// TIA Portal project "Övning 5" (V16)

(* hardware
DEVICE "S7-1200 station_1"  S7-1200 Station
   slot 0: "Rack_0"  S7-1200 Rack  Rack  V1.0
   slot 1: "PLC_1"  CPU 1212C DC/DC/DC  6ES7 212-1AE40-0XB0  V4.2
   slot 2: "DI 16x24VDC_1"  6ES7 221-1BH32-0XB0  V2.0
   slot 3: "DQ 16x24VDC_1"  SM 1222 DQ16 x 24VDC  6ES7 222-1BH32-0XB0  V2.0
*)

// ===== PLC "PLC_1"  CPU 1212C DC/DC/DC =====

VAR_GLOBAL   // PLC tag table "Default tag table"
   "ÅTERSTÄLLNING" AT %I0.0 : Bool;
   "VRED_MANUEL" AT %I0.1 : Bool;
   "VRED_AUTO" AT %I0.2 : Bool;
   "K_START" AT %I0.3 : Bool;
   "K_STOPP" AT %I0.4 : Bool;
   "K_PUMP1_TILL" AT %I0.5 : Bool;
   "K_PUMP1_FRÅN" AT %I0.6 : Bool;
   "K_PUMP2_TILL" AT %I8.0 : Bool;
   "K_PUMP2_FRÅN" AT %I8.1 : Bool;
   "K_VENTIL_STÄNG" AT %I8.2 : Bool;
   "K_VENTIL_ÖPPNA" AT %I8.3 : Bool;
   "K_LAMPTEST" AT %I8.4 : Bool;
   "NIVÅ_L6" AT %I9.0 : Bool;
   "NIVÅ_L5" AT %I9.1 : Bool;
   "NIVÅ_L4" AT %I9.2 : Bool;
   "NIVÅ_L3" AT %I9.3 : Bool;
   "NIVÅ_L2" AT %I9.4 : Bool;
   "NIVÅ_L1" AT %I9.5 : Bool;
   "MOTORSKYDD_B1" AT %I9.6 : Bool;
   "MOTORSKYDD_F2" AT %I9.7 : Bool;
   "L_ALARM" AT %Q12.0 : Bool;
   "L_PUMP1_TILL" AT %Q12.1 : Bool;
   "L_PUMP1_FRÅN" AT %Q12.2 : Bool;
   "L_VENTIL_ÖPPEN" AT %Q12.3 : Bool;
   "L_VENTIL_STÄNGD" AT %Q12.4 : Bool;
   "L_PUMP2_TILL" AT %Q12.5 : Bool;
   "L_PUMP2_FRÅN" AT %Q12.6 : Bool;
   "L_NIVÅ_ALARM" AT %Q12.7 : Bool;
   "KONTAKTOR_H" AT %Q13.0 : Bool;
   "KONTAKTOR_D" AT %Q13.1 : Bool;
   "KONTAKTOR_Y" AT %Q13.2 : Bool;
   "KONTAKTOR_DIREKT" AT %Q13.3 : Bool;
   "KONTAKTOR_MAGNETVENTIL" AT %Q13.4 : Bool;
   "KONTAKTOR_IND.VENTIL" AT %Q13.5 : Bool;
   "KONTAKTOR_BLIXT" AT %Q13.6 : Bool;
   "M_AUTO" AT %M0.0 : Bool;
   "M_MANUELL" AT %M0.1 : Bool;
   "M_VENTIL_ÖPPNA/STÄNG_MANU" AT %M0.2 : Bool;
   "M_PUMP1_TILL_MANUELL" AT %M0.3 : Bool;
   "M_PUMP2_TILL_MANUELL" AT %M0.4 : Bool;
   "M_VENTIL_ÖPPNA/STÄNG_AUTO" AT %M0.5 : Bool;
   "M_PUMP1_TILL_AUTO" AT %M0.6 : Bool;
   "M_PUMP2_TILL_AUTO" AT %M0.7 : Bool;
   "M_VARRANAN" AT %M1.0 : Bool;
   "M_BLIXT_AUTO" AT %M1.1 : Bool;
   "M_LARM_NIVÅ_AUTO" AT %M1.2 : Bool;
   "System_Byte" AT %MB1 : Byte;
   "Clock_Byte" AT %MB500 : Byte;
   "Clock_10Hz" AT %M500.0 : Bool;
   "Clock_5Hz" AT %M500.1 : Bool;
   "Clock_2.5Hz" AT %M500.2 : Bool;
   "Clock_2Hz" AT %M500.3 : Bool;
   "Clock_1.25Hz" AT %M500.4 : Bool;
   "Clock_1Hz" AT %M500.5 : Bool;
   "Clock_0.625Hz" AT %M500.6 : Bool;
   "Clock_0.5Hz" AT %M500.7 : Bool;
   "M_LARM_BLINKIE" AT %M2.0 : Bool;
   "M_LAMPTEST" AT %M2.1 : Bool;
   "M_LAMPTEST_AUTO" AT %M2.2 : Bool;
END_VAR

// folder: System blocks/Program resources

DATA_BLOCK "TIMER Y/D"   // DB1
{ S7_Optimized_Access := 'TRUE' }
AUTHOR : Simatic
FAMILY : IEC
NAME : IEC_TMR
VERSION : 1.0
// stored: InstanceOfName IEC_TIMER
"IEC_TIMER"
BEGIN
END_DATA_BLOCK

DATA_BLOCK "BLIXT-TIMER"   // DB2
{ S7_Optimized_Access := 'TRUE' }
AUTHOR : Simatic
FAMILY : IEC
NAME : IEC_TMR
VERSION : 1.0
// stored: InstanceOfName IEC_TIMER
"IEC_TIMER"
BEGIN
END_DATA_BLOCK

DATA_BLOCK "LAMP_TEST_AUTO"   // DB3
{ S7_Optimized_Access := 'TRUE' }
AUTHOR : Simatic
FAMILY : IEC
NAME : IEC_TMR
VERSION : 1.0
// stored: InstanceOfName IEC_TIMER
"IEC_TIMER"
BEGIN
END_DATA_BLOCK

// folder: (top level)

FUNCTION "Mongo" : Void   // FC1, LAD
{ S7_Optimized_Access := 'TRUE' }
VERSION : 0.1
   VAR_TEMP   // added for the SCL form of the ladder/FBD networks
      _w1 : Bool;
   END_VAR
BEGIN

REGION Network 1: MANUELL STARTKNAPP
   // Anläggningen startas med startknapp
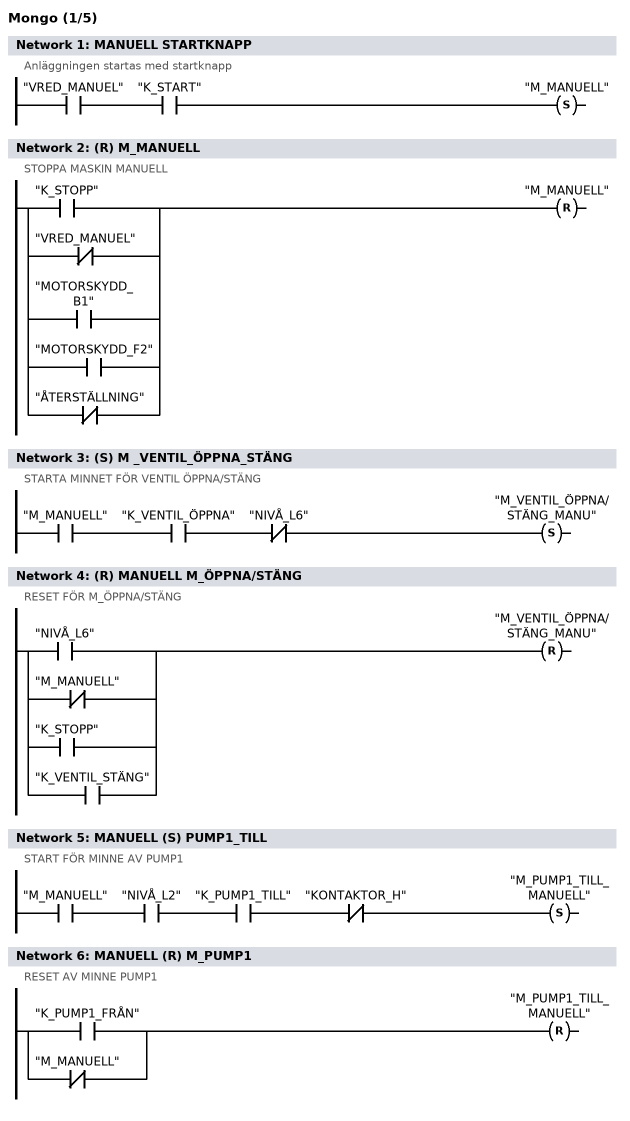
   RUNG wire#powerrail
      Contact( "VRED_MANUEL" )
      Contact( "K_START" )
      S_Coil( "M_MANUELL" )
   END_RUNG
   // the same network as SCL:
   IF "VRED_MANUEL" AND "K_START" THEN "M_MANUELL" := TRUE; END_IF;
END_REGION

REGION Network 2: (R) M_MANUELL
   // STOPPA MASKIN MANUELL
   RUNG wire#powerrail
      Contact( "K_STOPP" )
      wire#w1
      R_Coil( "M_MANUELL" )
   END_RUNG
   RUNG wire#powerrail
      I_Contact( "VRED_MANUEL" )
   END_RUNG wire#w1
   RUNG wire#powerrail
      Contact( "MOTORSKYDD_B1" )
   END_RUNG wire#w1
   RUNG wire#powerrail
      Contact( "MOTORSKYDD_F2" )
   END_RUNG wire#w1
   RUNG wire#powerrail
      I_Contact( "ÅTERSTÄLLNING" )
   END_RUNG wire#w1
   // the same network as SCL:
   IF "K_STOPP" OR NOT "VRED_MANUEL" OR "MOTORSKYDD_B1" OR "MOTORSKYDD_F2" OR NOT "ÅTERSTÄLLNING" THEN
       "M_MANUELL" := FALSE;
   END_IF;
END_REGION

REGION Network 3: (S) M _VENTIL_ÖPPNA_STÄNG
   // STARTA MINNET FÖR VENTIL ÖPPNA/STÄNG
   RUNG wire#powerrail
      Contact( "M_MANUELL" )
      Contact( "K_VENTIL_ÖPPNA" )
      I_Contact( "NIVÅ_L6" )
      S_Coil( "M_VENTIL_ÖPPNA/STÄNG_MANU" )
   END_RUNG
   // the same network as SCL:
   IF "M_MANUELL" AND "K_VENTIL_ÖPPNA" AND NOT "NIVÅ_L6" THEN "M_VENTIL_ÖPPNA/STÄNG_MANU" := TRUE; END_IF;
END_REGION

REGION Network 4: (R) MANUELL M_ÖPPNA/STÄNG
   // RESET FÖR M_ÖPPNA/STÄNG
   RUNG wire#powerrail
      Contact( "NIVÅ_L6" )
      wire#w1
      R_Coil( "M_VENTIL_ÖPPNA/STÄNG_MANU" )
   END_RUNG
   RUNG wire#powerrail
      I_Contact( "M_MANUELL" )
   END_RUNG wire#w1
   RUNG wire#powerrail
      Contact( "K_STOPP" )
   END_RUNG wire#w1
   RUNG wire#powerrail
      Contact( "K_VENTIL_STÄNG" )
   END_RUNG wire#w1
   // the same network as SCL:
   IF "NIVÅ_L6" OR NOT "M_MANUELL" OR "K_STOPP" OR "K_VENTIL_STÄNG" THEN
       "M_VENTIL_ÖPPNA/STÄNG_MANU" := FALSE;
   END_IF;
END_REGION

REGION Network 5: MANUELL (S) PUMP1_TILL
   // START FÖR MINNE AV PUMP1
   RUNG wire#powerrail
      Contact( "M_MANUELL" )
      Contact( "NIVÅ_L2" )
      Contact( "K_PUMP1_TILL" )
      I_Contact( "KONTAKTOR_H" )
      S_Coil( "M_PUMP1_TILL_MANUELL" )
   END_RUNG
   // the same network as SCL:
   IF "M_MANUELL" AND "NIVÅ_L2" AND "K_PUMP1_TILL" AND NOT "KONTAKTOR_H" THEN
       "M_PUMP1_TILL_MANUELL" := TRUE;
   END_IF;
END_REGION

REGION Network 6: MANUELL (R) M_PUMP1
   // RESET AV MINNE PUMP1
   RUNG wire#powerrail
      Contact( "K_PUMP1_FRÅN" )
      wire#w1
      R_Coil( "M_PUMP1_TILL_MANUELL" )
   END_RUNG
   RUNG wire#powerrail
      I_Contact( "M_MANUELL" )
   END_RUNG wire#w1
   // the same network as SCL:
   IF "K_PUMP1_FRÅN" OR NOT "M_MANUELL" THEN "M_PUMP1_TILL_MANUELL" := FALSE; END_IF;
END_REGION

REGION Network 7: MANUELL (S) M_PUMP2
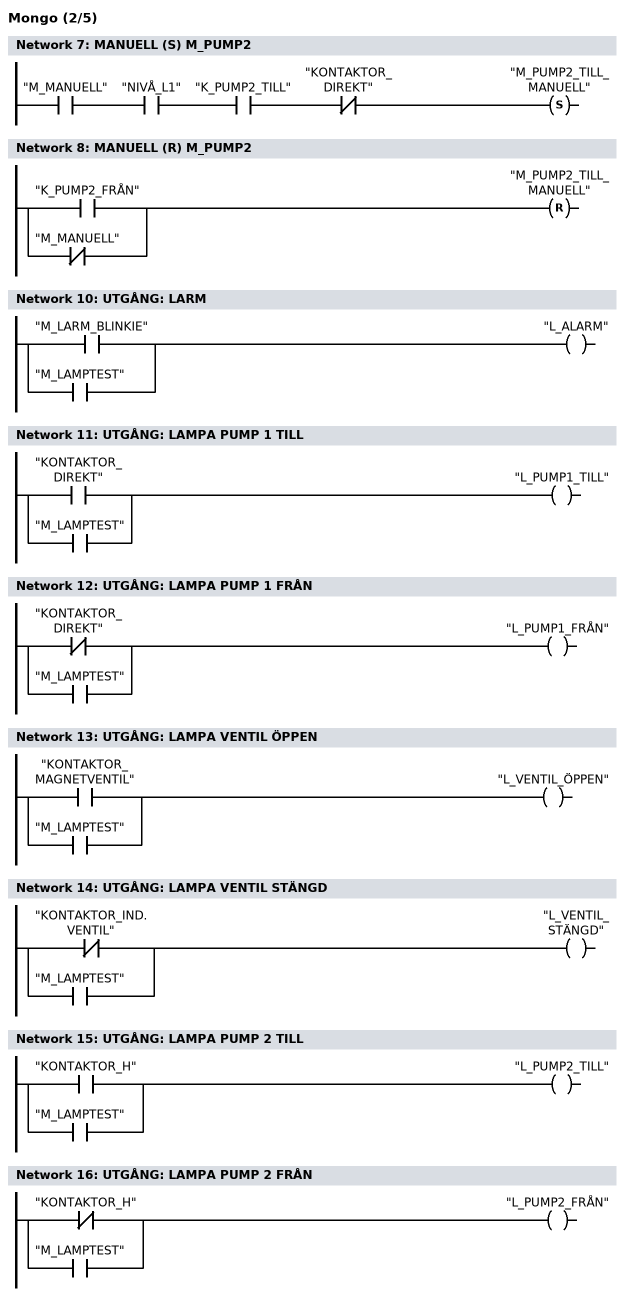
   RUNG wire#powerrail
      Contact( "M_MANUELL" )
      Contact( "NIVÅ_L1" )
      Contact( "K_PUMP2_TILL" )
      I_Contact( "KONTAKTOR_DIREKT" )
      S_Coil( "M_PUMP2_TILL_MANUELL" )
   END_RUNG
   // the same network as SCL:
   IF "M_MANUELL" AND "NIVÅ_L1" AND "K_PUMP2_TILL" AND NOT "KONTAKTOR_DIREKT" THEN
       "M_PUMP2_TILL_MANUELL" := TRUE;
   END_IF;
END_REGION

REGION Network 8: MANUELL (R) M_PUMP2
   RUNG wire#powerrail
      Contact( "K_PUMP2_FRÅN" )
      wire#w1
      R_Coil( "M_PUMP2_TILL_MANUELL" )
   END_RUNG
   RUNG wire#powerrail
      I_Contact( "M_MANUELL" )
   END_RUNG wire#w1
   // the same network as SCL:
   IF "K_PUMP2_FRÅN" OR NOT "M_MANUELL" THEN "M_PUMP2_TILL_MANUELL" := FALSE; END_IF;
END_REGION

REGION Network 10: UTGÅNG: LARM
   RUNG wire#powerrail
      Contact( "M_LARM_BLINKIE" )
      wire#w1
      Coil( "L_ALARM" )
   END_RUNG
   RUNG wire#powerrail
      Contact( "M_LAMPTEST" )
   END_RUNG wire#w1
   // the same network as SCL:
   "L_ALARM" := "M_LARM_BLINKIE" OR "M_LAMPTEST";
END_REGION

REGION Network 11: UTGÅNG: LAMPA PUMP 1 TILL
   RUNG wire#powerrail
      Contact( "KONTAKTOR_DIREKT" )
      wire#w1
      Coil( "L_PUMP1_TILL" )
   END_RUNG
   RUNG wire#powerrail
      Contact( "M_LAMPTEST" )
   END_RUNG wire#w1
   // the same network as SCL:
   "L_PUMP1_TILL" := "KONTAKTOR_DIREKT" OR "M_LAMPTEST";
END_REGION

REGION Network 12: UTGÅNG: LAMPA PUMP 1 FRÅN
   RUNG wire#powerrail
      I_Contact( "KONTAKTOR_DIREKT" )
      wire#w1
      Coil( "L_PUMP1_FRÅN" )
   END_RUNG
   RUNG wire#powerrail
      Contact( "M_LAMPTEST" )
   END_RUNG wire#w1
   // the same network as SCL:
   "L_PUMP1_FRÅN" := NOT "KONTAKTOR_DIREKT" OR "M_LAMPTEST";
END_REGION

REGION Network 13: UTGÅNG: LAMPA VENTIL ÖPPEN
   RUNG wire#powerrail
      Contact( "KONTAKTOR_MAGNETVENTIL" )
      wire#w1
      Coil( "L_VENTIL_ÖPPEN" )
   END_RUNG
   RUNG wire#powerrail
      Contact( "M_LAMPTEST" )
   END_RUNG wire#w1
   // the same network as SCL:
   "L_VENTIL_ÖPPEN" := "KONTAKTOR_MAGNETVENTIL" OR "M_LAMPTEST";
END_REGION

REGION Network 14: UTGÅNG: LAMPA VENTIL STÄNGD
   RUNG wire#powerrail
      I_Contact( "KONTAKTOR_IND.VENTIL" )
      wire#w1
      Coil( "L_VENTIL_STÄNGD" )
   END_RUNG
   RUNG wire#powerrail
      Contact( "M_LAMPTEST" )
   END_RUNG wire#w1
   // the same network as SCL:
   "L_VENTIL_STÄNGD" := NOT "KONTAKTOR_IND.VENTIL" OR "M_LAMPTEST";
END_REGION

REGION Network 15: UTGÅNG: LAMPA PUMP 2 TILL
   RUNG wire#powerrail
      Contact( "KONTAKTOR_H" )
      wire#w1
      Coil( "L_PUMP2_TILL" )
   END_RUNG
   RUNG wire#powerrail
      Contact( "M_LAMPTEST" )
   END_RUNG wire#w1
   // the same network as SCL:
   "L_PUMP2_TILL" := "KONTAKTOR_H" OR "M_LAMPTEST";
END_REGION

REGION Network 16: UTGÅNG: LAMPA PUMP 2 FRÅN
   RUNG wire#powerrail
      I_Contact( "KONTAKTOR_H" )
      wire#w1
      Coil( "L_PUMP2_FRÅN" )
   END_RUNG
   RUNG wire#powerrail
      Contact( "M_LAMPTEST" )
   END_RUNG wire#w1
   // the same network as SCL:
   "L_PUMP2_FRÅN" := NOT "KONTAKTOR_H" OR "M_LAMPTEST";
END_REGION

REGION Network 17: UTGÅNG: LAMPA NIVÅ LARM
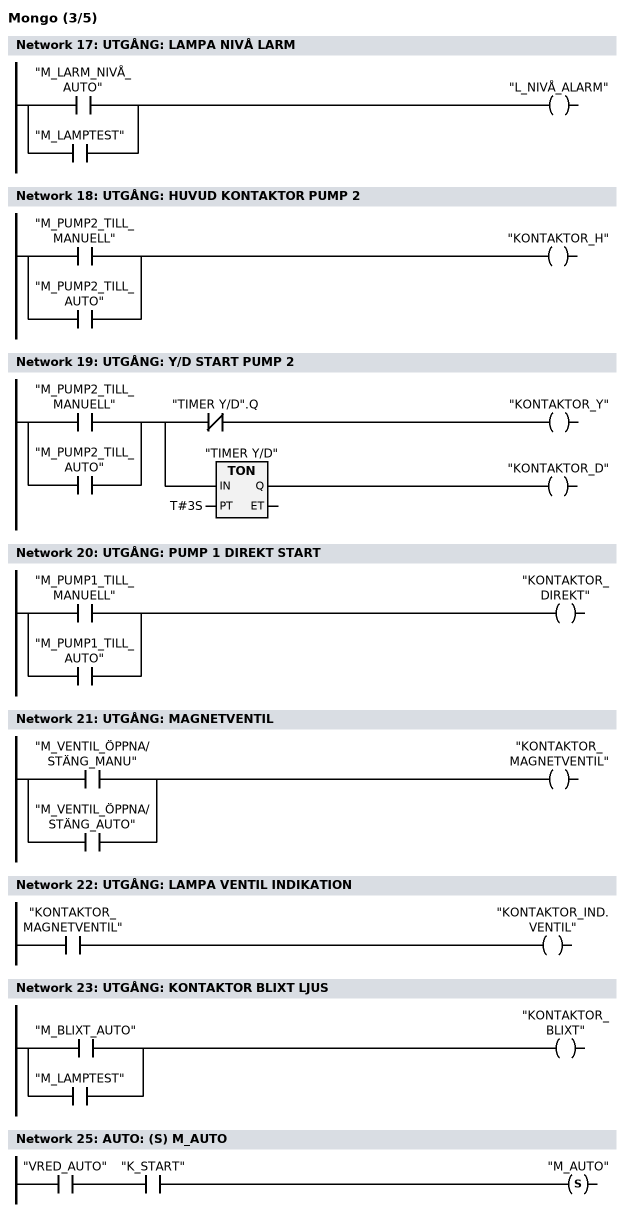
   RUNG wire#powerrail
      Contact( "M_LARM_NIVÅ_AUTO" )
      wire#w1
      Coil( "L_NIVÅ_ALARM" )
   END_RUNG
   RUNG wire#powerrail
      Contact( "M_LAMPTEST" )
   END_RUNG wire#w1
   // the same network as SCL:
   "L_NIVÅ_ALARM" := "M_LARM_NIVÅ_AUTO" OR "M_LAMPTEST";
END_REGION

REGION Network 18: UTGÅNG: HUVUD KONTAKTOR PUMP 2
   RUNG wire#powerrail
      Contact( "M_PUMP2_TILL_MANUELL" )
      wire#w1
      Coil( "KONTAKTOR_H" )
   END_RUNG
   RUNG wire#powerrail
      Contact( "M_PUMP2_TILL_AUTO" )
   END_RUNG wire#w1
   // the same network as SCL:
   "KONTAKTOR_H" := "M_PUMP2_TILL_MANUELL" OR "M_PUMP2_TILL_AUTO";
END_REGION

REGION Network 19: UTGÅNG: Y/D START PUMP 2
   #_w1 := "M_PUMP2_TILL_MANUELL" OR "M_PUMP2_TILL_AUTO";
   "KONTAKTOR_Y" := #_w1 AND NOT "TIMER Y/D".Q;
   "TIMER Y/D".TON(IN := #_w1, PT := T#3S);
   "KONTAKTOR_D" := "TIMER Y/D".Q;
END_REGION

REGION Network 20: UTGÅNG: PUMP 1 DIREKT START
   RUNG wire#powerrail
      Contact( "M_PUMP1_TILL_MANUELL" )
      wire#w1
      Coil( "KONTAKTOR_DIREKT" )
   END_RUNG
   RUNG wire#powerrail
      Contact( "M_PUMP1_TILL_AUTO" )
   END_RUNG wire#w1
   // the same network as SCL:
   "KONTAKTOR_DIREKT" := "M_PUMP1_TILL_MANUELL" OR "M_PUMP1_TILL_AUTO";
END_REGION

REGION Network 21: UTGÅNG: MAGNETVENTIL
   RUNG wire#powerrail
      Contact( "M_VENTIL_ÖPPNA/STÄNG_MANU" )
      wire#w1
      Coil( "KONTAKTOR_MAGNETVENTIL" )
   END_RUNG
   RUNG wire#powerrail
      Contact( "M_VENTIL_ÖPPNA/STÄNG_AUTO" )
   END_RUNG wire#w1
   // the same network as SCL:
   "KONTAKTOR_MAGNETVENTIL" := "M_VENTIL_ÖPPNA/STÄNG_MANU" OR "M_VENTIL_ÖPPNA/STÄNG_AUTO";
END_REGION

REGION Network 22: UTGÅNG: LAMPA VENTIL INDIKATION
   RUNG wire#powerrail
      Contact( "KONTAKTOR_MAGNETVENTIL" )
      Coil( "KONTAKTOR_IND.VENTIL" )
   END_RUNG
   // the same network as SCL:
   "KONTAKTOR_IND.VENTIL" := "KONTAKTOR_MAGNETVENTIL";
END_REGION

REGION Network 23: UTGÅNG: KONTAKTOR BLIXT LJUS
   RUNG wire#powerrail
      Contact( "M_BLIXT_AUTO" )
      wire#w1
      Coil( "KONTAKTOR_BLIXT" )
   END_RUNG
   RUNG wire#powerrail
      Contact( "M_LAMPTEST" )
   END_RUNG wire#w1
   // the same network as SCL:
   "KONTAKTOR_BLIXT" := "M_BLIXT_AUTO" OR "M_LAMPTEST";
END_REGION

REGION Network 25: AUTO: (S) M_AUTO
   RUNG wire#powerrail
      Contact( "VRED_AUTO" )
      Contact( "K_START" )
      S_Coil( "M_AUTO" )
   END_RUNG
   // the same network as SCL:
   IF "VRED_AUTO" AND "K_START" THEN "M_AUTO" := TRUE; END_IF;
END_REGION

REGION Network 26: AUTO: (R) M_AUTO
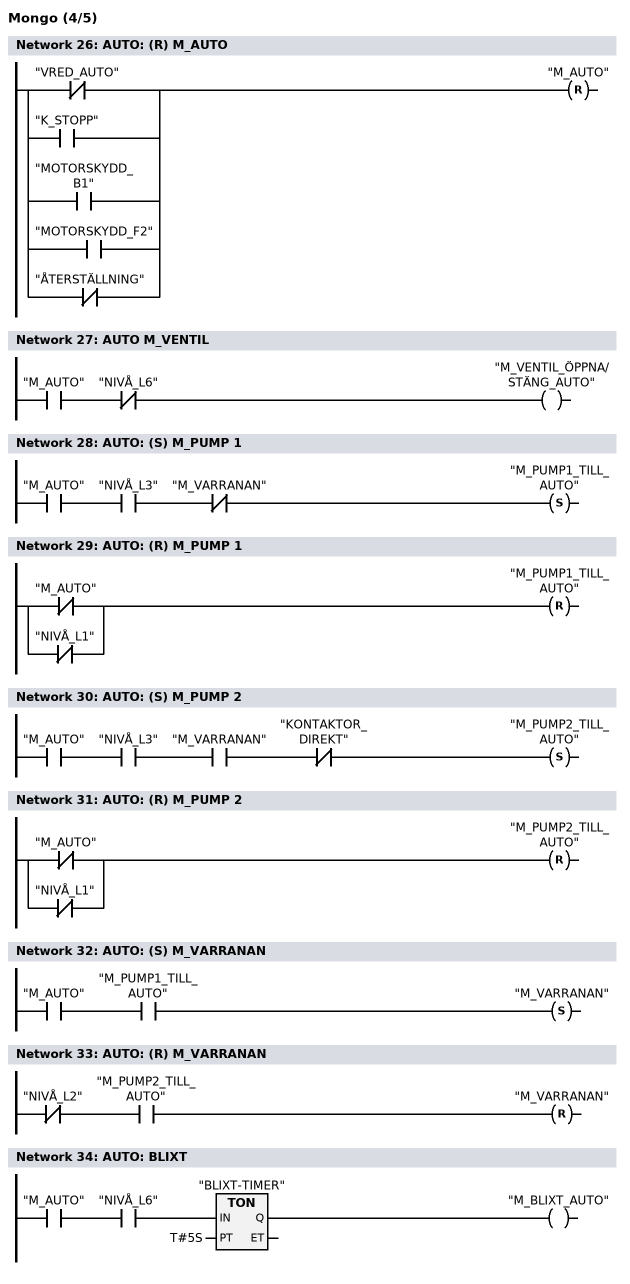
   RUNG wire#powerrail
      I_Contact( "VRED_AUTO" )
      wire#w1
      R_Coil( "M_AUTO" )
   END_RUNG
   RUNG wire#powerrail
      Contact( "K_STOPP" )
   END_RUNG wire#w1
   RUNG wire#powerrail
      Contact( "MOTORSKYDD_B1" )
   END_RUNG wire#w1
   RUNG wire#powerrail
      Contact( "MOTORSKYDD_F2" )
   END_RUNG wire#w1
   RUNG wire#powerrail
      I_Contact( "ÅTERSTÄLLNING" )
   END_RUNG wire#w1
   // the same network as SCL:
   IF NOT "VRED_AUTO" OR "K_STOPP" OR "MOTORSKYDD_B1" OR "MOTORSKYDD_F2" OR NOT "ÅTERSTÄLLNING" THEN
       "M_AUTO" := FALSE;
   END_IF;
END_REGION

REGION Network 27: AUTO M_VENTIL
   RUNG wire#powerrail
      Contact( "M_AUTO" )
      I_Contact( "NIVÅ_L6" )
      Coil( "M_VENTIL_ÖPPNA/STÄNG_AUTO" )
   END_RUNG
   // the same network as SCL:
   "M_VENTIL_ÖPPNA/STÄNG_AUTO" := "M_AUTO" AND NOT "NIVÅ_L6";
END_REGION

REGION Network 28: AUTO: (S) M_PUMP 1
   RUNG wire#powerrail
      Contact( "M_AUTO" )
      Contact( "NIVÅ_L3" )
      I_Contact( "M_VARRANAN" )
      S_Coil( "M_PUMP1_TILL_AUTO" )
   END_RUNG
   // the same network as SCL:
   IF "M_AUTO" AND "NIVÅ_L3" AND NOT "M_VARRANAN" THEN "M_PUMP1_TILL_AUTO" := TRUE; END_IF;
END_REGION

REGION Network 29: AUTO: (R) M_PUMP 1
   RUNG wire#powerrail
      I_Contact( "M_AUTO" )
      wire#w1
      R_Coil( "M_PUMP1_TILL_AUTO" )
   END_RUNG
   RUNG wire#powerrail
      I_Contact( "NIVÅ_L1" )
   END_RUNG wire#w1
   // the same network as SCL:
   IF NOT "M_AUTO" OR NOT "NIVÅ_L1" THEN "M_PUMP1_TILL_AUTO" := FALSE; END_IF;
END_REGION

REGION Network 30: AUTO: (S) M_PUMP 2
   RUNG wire#powerrail
      Contact( "M_AUTO" )
      Contact( "NIVÅ_L3" )
      Contact( "M_VARRANAN" )
      I_Contact( "KONTAKTOR_DIREKT" )
      S_Coil( "M_PUMP2_TILL_AUTO" )
   END_RUNG
   // the same network as SCL:
   IF "M_AUTO" AND "NIVÅ_L3" AND "M_VARRANAN" AND NOT "KONTAKTOR_DIREKT" THEN
       "M_PUMP2_TILL_AUTO" := TRUE;
   END_IF;
END_REGION

REGION Network 31: AUTO: (R) M_PUMP 2
   RUNG wire#powerrail
      I_Contact( "M_AUTO" )
      wire#w1
      R_Coil( "M_PUMP2_TILL_AUTO" )
   END_RUNG
   RUNG wire#powerrail
      I_Contact( "NIVÅ_L1" )
   END_RUNG wire#w1
   // the same network as SCL:
   IF NOT "M_AUTO" OR NOT "NIVÅ_L1" THEN "M_PUMP2_TILL_AUTO" := FALSE; END_IF;
END_REGION

REGION Network 32: AUTO: (S) M_VARRANAN
   RUNG wire#powerrail
      Contact( "M_AUTO" )
      Contact( "M_PUMP1_TILL_AUTO" )
      S_Coil( "M_VARRANAN" )
   END_RUNG
   // the same network as SCL:
   IF "M_AUTO" AND "M_PUMP1_TILL_AUTO" THEN "M_VARRANAN" := TRUE; END_IF;
END_REGION

REGION Network 33: AUTO: (R) M_VARRANAN
   RUNG wire#powerrail
      I_Contact( "NIVÅ_L2" )
      Contact( "M_PUMP2_TILL_AUTO" )
      R_Coil( "M_VARRANAN" )
   END_RUNG
   // the same network as SCL:
   IF NOT "NIVÅ_L2" AND "M_PUMP2_TILL_AUTO" THEN "M_VARRANAN" := FALSE; END_IF;
END_REGION

REGION Network 34: AUTO: BLIXT
   "BLIXT-TIMER".TON(IN := "M_AUTO" AND "NIVÅ_L6", PT := T#5S);
   "M_BLIXT_AUTO" := "BLIXT-TIMER".Q;
END_REGION

REGION Network 35: AUTO: (S) M_LARM_NIVÅ
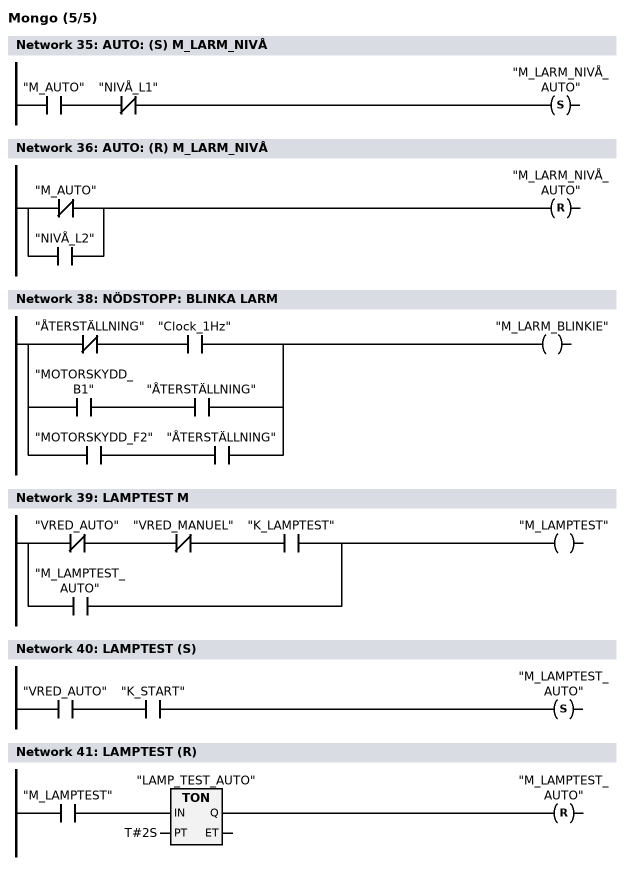
   RUNG wire#powerrail
      Contact( "M_AUTO" )
      I_Contact( "NIVÅ_L1" )
      S_Coil( "M_LARM_NIVÅ_AUTO" )
   END_RUNG
   // the same network as SCL:
   IF "M_AUTO" AND NOT "NIVÅ_L1" THEN "M_LARM_NIVÅ_AUTO" := TRUE; END_IF;
END_REGION

REGION Network 36: AUTO: (R) M_LARM_NIVÅ
   RUNG wire#powerrail
      I_Contact( "M_AUTO" )
      wire#w1
      R_Coil( "M_LARM_NIVÅ_AUTO" )
   END_RUNG
   RUNG wire#powerrail
      Contact( "NIVÅ_L2" )
   END_RUNG wire#w1
   // the same network as SCL:
   IF NOT "M_AUTO" OR "NIVÅ_L2" THEN "M_LARM_NIVÅ_AUTO" := FALSE; END_IF;
END_REGION

REGION Network 38: NÖDSTOPP: BLINKA LARM
   RUNG wire#powerrail
      I_Contact( "ÅTERSTÄLLNING" )
      Contact( "Clock_1Hz" )
      wire#w1
      Coil( "M_LARM_BLINKIE" )
   END_RUNG
   RUNG wire#powerrail
      Contact( "MOTORSKYDD_B1" )
      Contact( "ÅTERSTÄLLNING" )
   END_RUNG wire#w1
   RUNG wire#powerrail
      Contact( "MOTORSKYDD_F2" )
      Contact( "ÅTERSTÄLLNING" )
   END_RUNG wire#w1
   // the same network as SCL:
   "M_LARM_BLINKIE" := (NOT "ÅTERSTÄLLNING" AND "Clock_1Hz") OR ("MOTORSKYDD_B1" AND "ÅTERSTÄLLNING") OR ("MOTORSKYDD_F2" AND "ÅTERSTÄLLNING");
END_REGION

REGION Network 39: LAMPTEST M
   RUNG wire#powerrail
      I_Contact( "VRED_AUTO" )
      I_Contact( "VRED_MANUEL" )
      Contact( "K_LAMPTEST" )
      wire#w1
      Coil( "M_LAMPTEST" )
   END_RUNG
   RUNG wire#powerrail
      Contact( "M_LAMPTEST_AUTO" )
   END_RUNG wire#w1
   // the same network as SCL:
   "M_LAMPTEST" := (NOT "VRED_AUTO" AND NOT "VRED_MANUEL" AND "K_LAMPTEST") OR "M_LAMPTEST_AUTO";
END_REGION

REGION Network 40: LAMPTEST (S)
   RUNG wire#powerrail
      Contact( "VRED_AUTO" )
      Contact( "K_START" )
      S_Coil( "M_LAMPTEST_AUTO" )
   END_RUNG
   // the same network as SCL:
   IF "VRED_AUTO" AND "K_START" THEN "M_LAMPTEST_AUTO" := TRUE; END_IF;
END_REGION

REGION Network 41: LAMPTEST (R)
   "LAMP_TEST_AUTO".TON(IN := "M_LAMPTEST", PT := T#2S);
   IF "LAMP_TEST_AUTO".Q THEN "M_LAMPTEST_AUTO" := FALSE; END_IF;
END_REGION
END_FUNCTION

ORGANIZATION_BLOCK "Main"   // OB1, LAD, ProgramCycle
TITLE = "Main Program Sweep (Cycle)"
{ S7_Optimized_Access := 'TRUE' }
VERSION : 0.1
   VAR_INPUT
      Initial_Call : Bool;   // Initial call of this OB
      Remanence : Bool;   // =True, if remanent data are available
   END_VAR
BEGIN

REGION Network 1
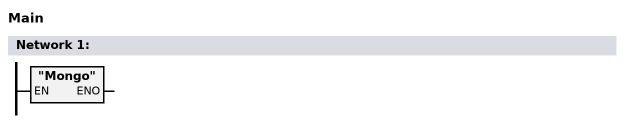
   RUNG wire#powerrail
      "Mongo"()
   END_RUNG
   // the same network as SCL:
   "Mongo"();
END_REGION
END_ORGANIZATION_BLOCK